FUNCTION F_DateNow : STRING
VAR_INPUT
END_VAR
VAR
END_VAR

F_DateNow := LEFT(GVL_General.DateTimeNow,10);

END_FUNCTION

(* stored: Version 1.1.0.1, ProductVersion 3.1.4022.16
   POU F_DateNow: Id {f460680d-b61c-46b3-848a-8544b3c7f190}, SpecialFunc None *)
